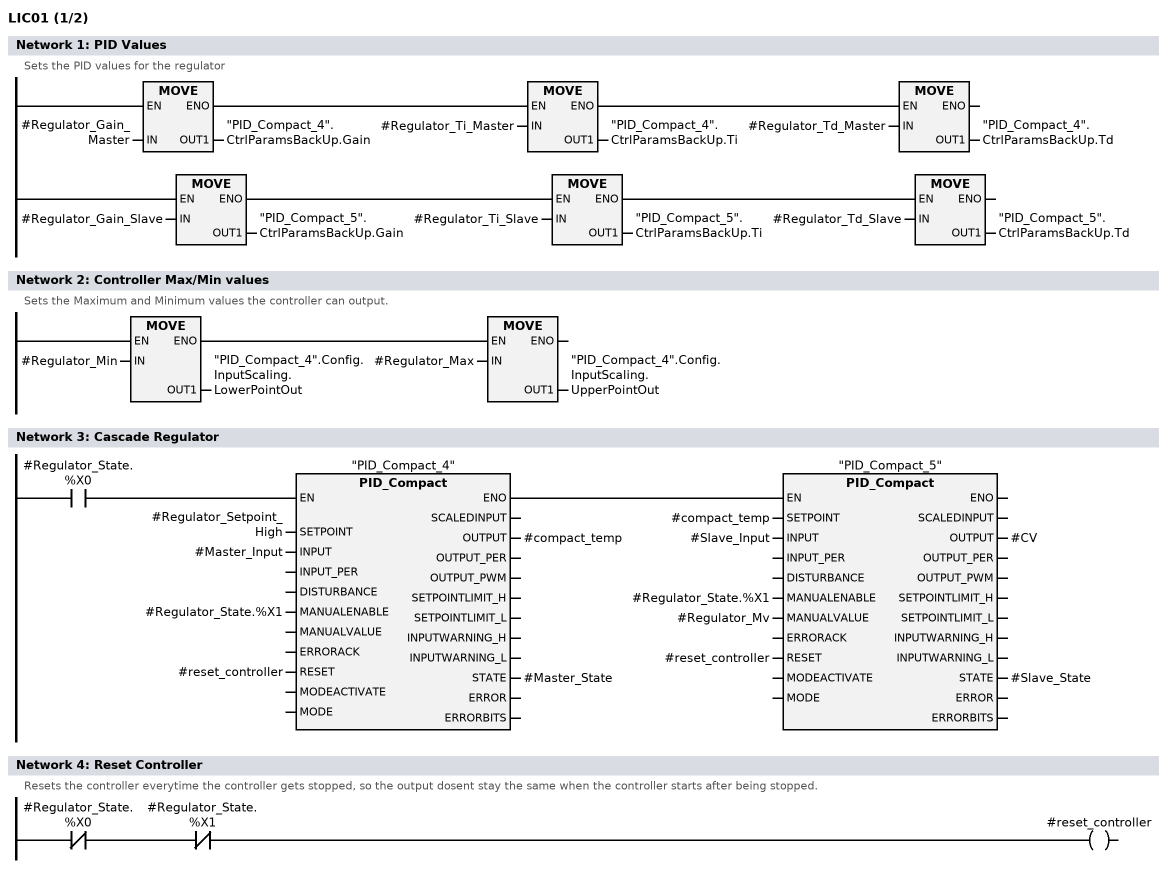
   RUNG wire#powerrail
      Move(in := #Regulator_Gain_Master, out1 => "PID_Compact_4".CtrlParamsBackUp.Gain)
      Move(in := #Regulator_Ti_Master, out1 => "PID_Compact_4".CtrlParamsBackUp.Ti)
      Move(in := #Regulator_Td_Master, out1 => "PID_Compact_4".CtrlParamsBackUp.Td)
   END_RUNG
   RUNG wire#powerrail
      Move(in := #Regulator_Gain_Slave, out1 => "PID_Compact_5".CtrlParamsBackUp.Gain)
      Move(in := #Regulator_Ti_Slave, out1 => "PID_Compact_5".CtrlParamsBackUp.Ti)
      Move(in := #Regulator_Td_Slave, out1 => "PID_Compact_5".CtrlParamsBackUp.Td)
   END_RUNG
   // the same network as SCL:
   "PID_Compact_4".CtrlParamsBackUp.Gain := #Regulator_Gain_Master;
   "PID_Compact_4".CtrlParamsBackUp.Ti := #Regulator_Ti_Master;
   "PID_Compact_4".CtrlParamsBackUp.Td := #Regulator_Td_Master;
   "PID_Compact_5".CtrlParamsBackUp.Gain := #Regulator_Gain_Slave;
   "PID_Compact_5".CtrlParamsBackUp.Ti := #Regulator_Ti_Slave;
   "PID_Compact_5".CtrlParamsBackUp.Td := #Regulator_Td_Slave;
END_REGION

REGION Network 2: Controller Max/Min values
   // Sets the Maximum and Minimum values the controller can output.
   RUNG wire#powerrail
      Move(in := #Regulator_Min, out1 => "PID_Compact_4".Config.InputScaling.LowerPointOut)
      Move(in := #Regulator_Max, out1 => "PID_Compact_4".Config.InputScaling.UpperPointOut)
   END_RUNG
   // the same network as SCL:
   "PID_Compact_4".Config.InputScaling.LowerPointOut := #Regulator_Min;
   "PID_Compact_4".Config.InputScaling.UpperPointOut := #Regulator_Max;
END_REGION

REGION Network 3: Cascade Regulator
   // ENO of a box is taken as its EN; it also drops when the box reports an error
   IF #Regulator_State.%X0 THEN
       "PID_Compact_4"(Setpoint := #Regulator_Setpoint_High,   // PID_Compact
                       Input := #Master_Input,
                       ManualEnable := #Regulator_State.%X1,
                       Reset := #reset_controller,
                       Output => #compact_temp,
                       State => #Master_State);
       "PID_Compact_5"(Setpoint := #compact_temp,   // PID_Compact
                       Input := #Slave_Input,
                       ManualEnable := #Regulator_State.%X1,
                       ManualValue := #Regulator_Mv,
                       Reset := #reset_controller,
                       Output => #CV,
                       State => #Slave_State);
   END_IF;
END_REGION

REGION Network 4: Reset Controller
   // Resets the controller everytime the controller gets stopped, so the output dosent stay the same when the controller starts after being stopped.
   RUNG wire#powerrail
      I_Contact( #Regulator_State.%X0 )
      I_Contact( #Regulator_State.%X1 )
      Coil( #reset_controller )
   END_RUNG
   // the same network as SCL:
   #reset_controller := NOT #Regulator_State.%X0 AND NOT #Regulator_State.%X1;
END_REGION

REGION Network 5: Controller Status
   // Sets different bits in the alarm word and forwards it.
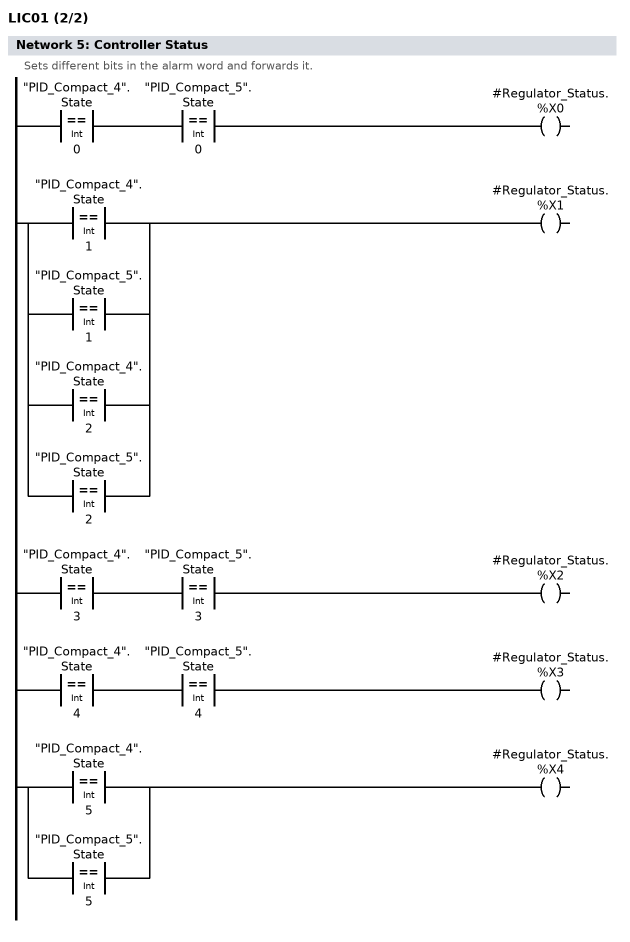
   RUNG wire#powerrail
      { S7_Templates := "SrcType := Int" } EQ_Contact(in1 := "PID_Compact_4".State, in2 := 0)
      { S7_Templates := "SrcType := Int" } EQ_Contact(in1 := "PID_Compact_5".State, in2 := 0)
      Coil( #Regulator_Status.%X0 )
   END_RUNG
   RUNG wire#powerrail
      { S7_Templates := "SrcType := Int" } EQ_Contact(in1 := "PID_Compact_4".State, in2 := 1)
      wire#w1
      Coil( #Regulator_Status.%X1 )
   END_RUNG
   RUNG wire#powerrail
      { S7_Templates := "SrcType := Int" } EQ_Contact(in1 := "PID_Compact_5".State, in2 := 1)
   END_RUNG wire#w1
   RUNG wire#powerrail
      { S7_Templates := "SrcType := Int" } EQ_Contact(in1 := "PID_Compact_4".State, in2 := 2)
   END_RUNG wire#w1
   RUNG wire#powerrail
      { S7_Templates := "SrcType := Int" } EQ_Contact(in1 := "PID_Compact_5".State, in2 := 2)
   END_RUNG wire#w1
   RUNG wire#powerrail
      { S7_Templates := "SrcType := Int" } EQ_Contact(in1 := "PID_Compact_4".State, in2 := 3)
      { S7_Templates := "SrcType := Int" } EQ_Contact(in1 := "PID_Compact_5".State, in2 := 3)
      Coil( #Regulator_Status.%X2 )
   END_RUNG
   RUNG wire#powerrail
      { S7_Templates := "SrcType := Int" } EQ_Contact(in1 := "PID_Compact_4".State, in2 := 4)
      { S7_Templates := "SrcType := Int" } EQ_Contact(in1 := "PID_Compact_5".State, in2 := 4)
      Coil( #Regulator_Status.%X3 )
   END_RUNG
   RUNG wire#powerrail
      { S7_Templates := "SrcType := Int" } EQ_Contact(in1 := "PID_Compact_4".State, in2 := 5)
      wire#w2
      Coil( #Regulator_Status.%X4 )
   END_RUNG
   RUNG wire#powerrail
      { S7_Templates := "SrcType := Int" } EQ_Contact(in1 := "PID_Compact_5".State, in2 := 5)
   END_RUNG wire#w2
   // the same network as SCL:
   #Regulator_Status.%X0 := ("PID_Compact_4".State = 0) AND ("PID_Compact_5".State = 0);
   #Regulator_Status.%X1 := ("PID_Compact_4".State = 1) OR ("PID_Compact_5".State = 1) OR ("PID_Compact_4".State = 2) OR ("PID_Compact_5".State = 2);
   #Regulator_Status.%X2 := ("PID_Compact_4".State = 3) AND ("PID_Compact_5".State = 3);
   #Regulator_Status.%X3 := ("PID_Compact_4".State = 4) AND ("PID_Compact_5".State = 4);
   #Regulator_Status.%X4 := ("PID_Compact_4".State = 5) OR ("PID_Compact_5".State = 5);
END_REGION
END_FUNCTION_BLOCK

// ===== library: MasterCopy "TRANSMITTER" =====

// folder: Scaling

FUNCTION_BLOCK "LT01"   // FB2, LAD
{ S7_Optimized_Access := 'FALSE' }
VERSION : 0.1
   VAR_INPUT
      t_sp_hh : Int;   // transmitter setpoint high-high
      t_sp_h : Int;   // transmitter setpoint high
      t_sp_l : Int;   // transmitter setpoint low
      t_sp_ll : Int;   // transmitter setpoint low-low
      t_sp_scale_high : Int;   // transmitter setpoint scale high
      t_sp_scale_low : Int;   // transmitter setpoint scale low
      t_hys : Int;   // transmitter hysteresis
      t_val : Int;   // transmitter value
   END_VAR
   VAR_OUTPUT
      t_pv : Real;   // transmitter process value
      t_aw : Int;   // transmitter alarm word
      t_alarm : Bool;   // transmitter alarm bool
   END_VAR
   VAR_TEMP
      t_temp : Real;
      t_pv_temp : Int;
   END_VAR
BEGIN

REGION Network 1
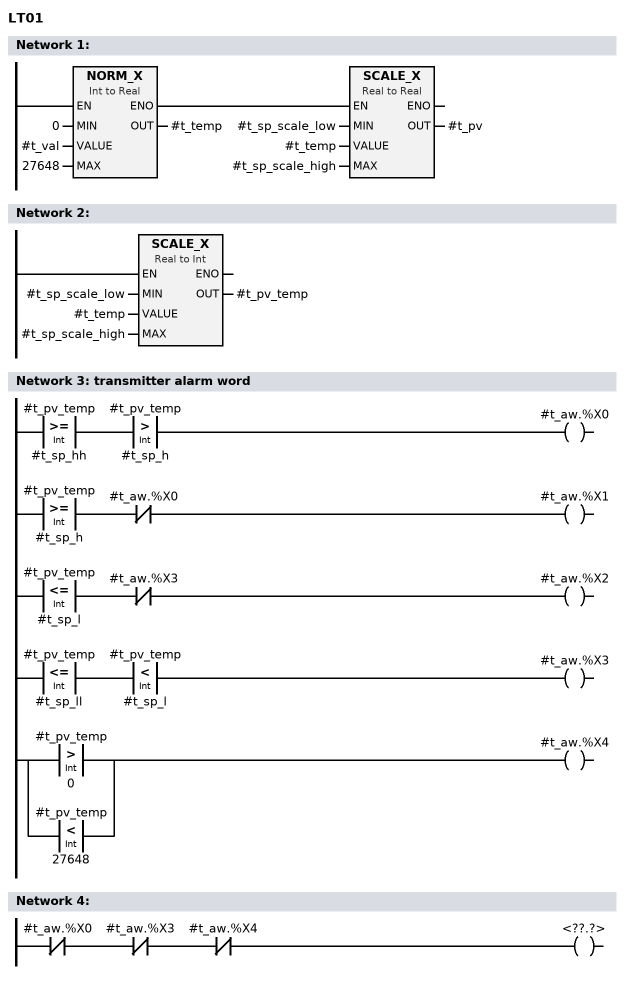
   RUNG wire#powerrail
      { S7_Templates := "[SrcType := Int, DestType := Real]"; S7_GenerateENO := "TRUE" } Normalize(min := 0, value := #t_val, max := 27648, out => #t_temp)
      { S7_Templates := "[SrcType := Real, DestType := Real]"; S7_GenerateENO := "TRUE" } Scale(min := #t_sp_scale_low, value := #t_temp, max := #t_sp_scale_high, out => #t_pv)
   END_RUNG
   // the same network as SCL:
   // ENO of a box is taken as its EN; it also drops when the box reports an error
   #t_temp := NORM_X(MIN := 0, VALUE := #t_val, MAX := 27648);
   #t_pv := SCALE_X(MIN := #t_sp_scale_low, VALUE := #t_temp, MAX := #t_sp_scale_high);
END_REGION

REGION Network 2
   RUNG wire#powerrail
      { S7_Templates := "[SrcType := Real, DestType := Int]"; S7_GenerateENO := "TRUE" } Scale(min := #t_sp_scale_low, value := #t_temp, max := #t_sp_scale_high, out => #t_pv_temp)
   END_RUNG
   // the same network as SCL:
   #t_pv_temp := SCALE_X(MIN := #t_sp_scale_low, VALUE := #t_temp, MAX := #t_sp_scale_high);
END_REGION

REGION Network 3: transmitter alarm word
   RUNG wire#powerrail
      { S7_Templates := "SrcType := Int" } GE_Contact(in1 := #t_pv_temp, in2 := #t_sp_hh)
      { S7_Templates := "SrcType := Int" } GT_Contact(in1 := #t_pv_temp, in2 := #t_sp_h)
      Coil( #t_aw.%X0 )
   END_RUNG
   RUNG wire#powerrail
      { S7_Templates := "SrcType := Int" } GE_Contact(in1 := #t_pv_temp, in2 := #t_sp_h)
      I_Contact( #t_aw.%X0 )
      Coil( #t_aw.%X1 )
   END_RUNG
   RUNG wire#powerrail
      { S7_Templates := "SrcType := Int" } LE_Contact(in1 := #t_pv_temp, in2 := #t_sp_l)
      I_Contact( #t_aw.%X3 )
      Coil( #t_aw.%X2 )
   END_RUNG
   RUNG wire#powerrail
      { S7_Templates := "SrcType := Int" } LE_Contact(in1 := #t_pv_temp, in2 := #t_sp_ll)
      { S7_Templates := "SrcType := Int" } LT_Contact(in1 := #t_pv_temp, in2 := #t_sp_l)
      Coil( #t_aw.%X3 )
   END_RUNG
   RUNG wire#powerrail
      { S7_Templates := "SrcType := Int" } GT_Contact(in1 := #t_pv_temp, in2 := 0)
      wire#w1
      Coil( #t_aw.%X4 )
   END_RUNG
   RUNG wire#powerrail
      { S7_Templates := "SrcType := Int" } LT_Contact(in1 := #t_pv_temp, in2 := 27648)
   END_RUNG wire#w1
   // the same network as SCL:
   #t_aw.%X0 := (#t_pv_temp >= #t_sp_hh) AND (#t_pv_temp > #t_sp_h);
   #t_aw.%X1 := (#t_pv_temp >= #t_sp_h) AND NOT #t_aw.%X0;
   #t_aw.%X2 := (#t_pv_temp <= #t_sp_l) AND NOT #t_aw.%X3;
   #t_aw.%X3 := (#t_pv_temp <= #t_sp_ll) AND (#t_pv_temp < #t_sp_l);
   #t_aw.%X4 := (#t_pv_temp > 0) OR (#t_pv_temp < 27648);
END_REGION

REGION Network 4
   RUNG wire#powerrail
      I_Contact( #t_aw.%X0 )
      I_Contact( #t_aw.%X3 )
      I_Contact( #t_aw.%X4 )
      Coil(  )
   END_RUNG
   // the same network as SCL:
   <??.?> := NOT #t_aw.%X0 AND NOT #t_aw.%X3 AND NOT #t_aw.%X4;
END_REGION
END_FUNCTION_BLOCK